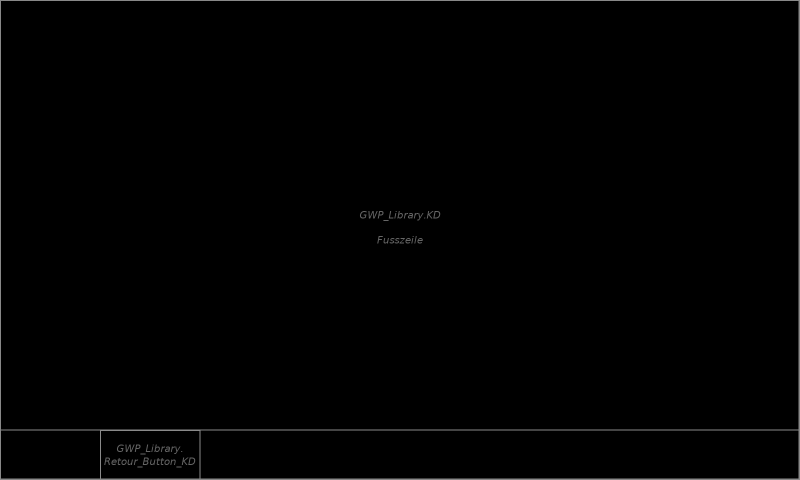
VISUALIZATION KD  // 800x480
    Frame (0,0 800x480)
        shows Fusszeile()
    Frame (100,430 100x50)
        shows GWP_Library.Retour_Button_KD()
    Frame (0,0 800x430)
        shows GWP_Library.KD(FB_KD := MAIN.KD_0)
END_VISUALIZATION

(* stored: Version 1.1.0.1, ProductVersion 3.1.4022.6
   Visu KD: Id {aae19a2c-7e8d-481f-b93a-3465f9c816f7} *)
